ABB RAPID module: Module1.mod

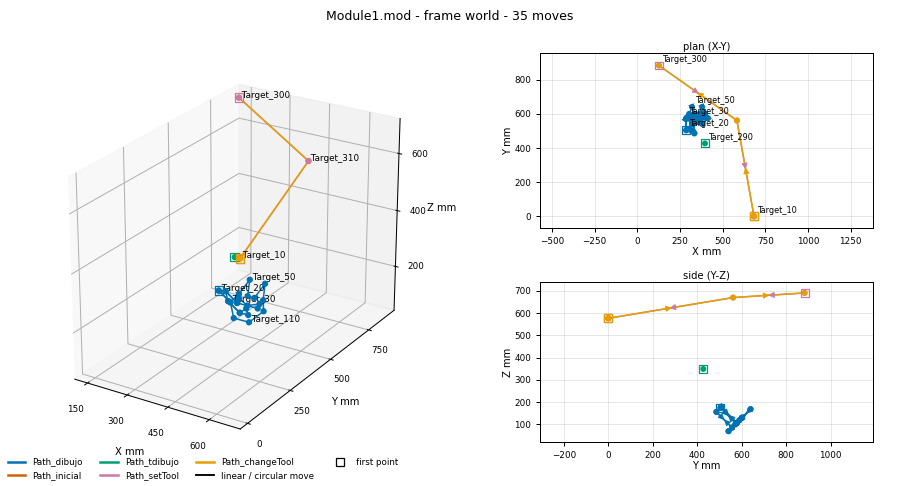
[picture p0: tool path of Module1.mod in frame world, 35 of 35 moves have a stored position in this frame; points joined in program order, loops and branches not executed]
MODULE Module1
        CONST robtarget Target_20:=[[-143.869244178,87.031135529,-100.000191842],[0.335710695,0,0,-0.941965142],[0,0,0,0],[9E+09,9E+09,9E+09,9E+09,9E+09,9E+09]];
    CONST robtarget Target_30:=[[-143.869244206,87.031135529,-0.000191841],[0.335710695,0,0,-0.941965142],[0,0,0,0],[9E+09,9E+09,9E+09,9E+09,9E+09,9E+09]];
    CONST robtarget Target_40:=[[-108.026112862,104.235837146,-0.000191832],[0.335710695,0,0,-0.941965142],[0,0,0,0],[9E+09,9E+09,9E+09,9E+09,9E+09,9E+09]];
    CONST robtarget Target_50:=[[-52.110827945,121.440538768,-0.000191815],[0.335710694,0,0.000000001,-0.941965143],[0,0,0,0],[9E+09,9E+09,9E+09,9E+09,9E+09,9E+09]];
    CONST robtarget Target_60:=[[-108.026112855,137.808909158,-0.000191832],[0.335710694,0,0.000000001,-0.941965143],[0,0,0,0],[9E+09,9E+09,9E+09,9E+09,9E+09,9E+09]];
    CONST robtarget Target_70:=[[-108.026112855,163.915610617,-0.000191832],[0.335710695,0,0,-0.941965142],[0,0,0,0],[9E+09,9E+09,9E+09,9E+09,9E+09,9E+09]];
    CONST robtarget Target_80:=[[-52.110827945,180.283981007,-0.000191815],[0.335710695,0,-0.000000001,-0.941965142],[0,0,0,0],[9E+09,9E+09,9E+09,9E+09,9E+09,9E+09]];
    CONST robtarget Target_90:=[[-108.026112862,197.48868263,-0.000191832],[0.335710695,0,-0.000000001,-0.941965142],[0,0,0,0],[9E+09,9E+09,9E+09,9E+09,9E+09,9E+09]];
    CONST robtarget Target_100:=[[-143.869244206,214.693384246,-0.000191841],[0.335710695,0,0,-0.941965142],[0,0,0,0],[9E+09,9E+09,9E+09,9E+09,9E+09,9E+09]];
    CONST robtarget Target_110:=[[-192.615902843,180.283981007,-0.000191856],[0.335710695,0,0,-0.941965142],[0,0,0,0],[9E+09,9E+09,9E+09,9E+09,9E+09,9E+09]];
    CONST robtarget Target_120:=[[-192.615902844,121.440538769,-0.000191855],[0.335710695,0,0,-0.941965142],[0,0,0,0],[9E+09,9E+09,9E+09,9E+09,9E+09,9E+09]];
    CONST robtarget Target_130:=[[-143.869244206,87.031135529,-0.000191841],[0.335710695,0,0,-0.941965142],[0,0,0,0],[9E+09,9E+09,9E+09,9E+09,9E+09,9E+09]];
    CONST robtarget Target_140:=[[-143.869244178,87.031135529,-100.000191842],[0.335710695,0,0,-0.941965142],[0,0,0,0],[9E+09,9E+09,9E+09,9E+09,9E+09,9E+09]];
    CONST robtarget Target_150:=[[-139.856817565,111.33818796,-100.000191841],[0.335710706,0,0,-0.941965138],[0,0,0,0],[9E+09,9E+09,9E+09,9E+09,9E+09,9E+09]];
    CONST robtarget Target_160:=[[-139.856817593,111.33818796,-0.00019184],[0.335710706,0,0,-0.941965138],[0,0,0,0],[9E+09,9E+09,9E+09,9E+09,9E+09,9E+09]];
    CONST robtarget Target_170:=[[-123.434971754,111.33818796,-0.000191836],[0.335710706,0,0,-0.941965138],[0,0,0,0],[9E+09,9E+09,9E+09,9E+09,9E+09,9E+09]];
    CONST robtarget Target_180:=[[-139.282664103,150.862259888,-0.000191841],[0.335710706,-0.000000001,-0.000000001,-0.941965138],[0,0,0,0],[9E+09,9E+09,9E+09,9E+09,9E+09,9E+09]];
    CONST robtarget Target_190:=[[-123.434971754,190.386331815,-0.000191836],[0.335710706,0,0.000000001,-0.941965138],[0,0,0,0],[9E+09,9E+09,9E+09,9E+09,9E+09,9E+09]];
    CONST robtarget Target_200:=[[-139.856817593,190.386331815,-0.00019184],[0.335710706,0,0,-0.941965138],[0,0,0,0],[9E+09,9E+09,9E+09,9E+09,9E+09,9E+09]];
    CONST robtarget Target_210:=[[-139.856817593,111.33818796,-0.00019184],[0.335710706,0,0,-0.941965138],[0,0,0,0],[9E+09,9E+09,9E+09,9E+09,9E+09,9E+09]];
    CONST robtarget Target_220:=[[-139.856817565,111.33818796,-100.000191841],[0.335710706,0,0,-0.941965138],[0,0,0,0],[9E+09,9E+09,9E+09,9E+09,9E+09,9E+09]];
    CONST robtarget Target_230:=[[-169.742573497,134.622057219,-100.000191849],[0.335710706,0,0,-0.941965138],[0,0,0,0],[9E+09,9E+09,9E+09,9E+09,9E+09,9E+09]];
    CONST robtarget Target_240:=[[-169.742573525,134.622057219,-0.000191849],[0.335710706,0,0,-0.941965138],[0,0,0,0],[9E+09,9E+09,9E+09,9E+09,9E+09,9E+09]];
    CONST robtarget Target_250:=[[-150.103708423,150.862259887,-0.000191843],[0.335710706,0,0,-0.941965138],[0,0,0,0],[9E+09,9E+09,9E+09,9E+09,9E+09,9E+09]];
    CONST robtarget Target_260:=[[-169.742573525,167.102462557,-0.000191849],[0.335710706,0,0,-0.941965138],[0,0,0,0],[9E+09,9E+09,9E+09,9E+09,9E+09,9E+09]];
    CONST robtarget Target_270:=[[-169.742573525,134.622057219,-0.000191849],[0.335710706,0,0,-0.941965138],[0,0,0,0],[9E+09,9E+09,9E+09,9E+09,9E+09,9E+09]];
    CONST robtarget Target_280:=[[-169.742573497,134.622057219,-100.000191849],[0.335710706,0,0,-0.941965138],[0,0,0,0],[9E+09,9E+09,9E+09,9E+09,9E+09,9E+09]];
    CONST robtarget Target_10:=[[683.826857055,0,576.999996593],[0.499999994,0,0.866025407,0],[0,0,0,0],[9E+09,9E+09,9E+09,9E+09,9E+09,9E+09]];
    CONST robtarget Target_290:=[[396.786283568,427.182015311,348.94513545],[0.291756838,-0.37886731,0.868997985,0.127200673],[0,0,-1,0],[9E+09,9E+09,9E+09,9E+09,9E+09,9E+09]];
    CONST robtarget Target_300:=[[127.426507212,883.161303543,691.12368836],[0.534755638,-0.462711495,0.534265162,0.463136282],[0,0,-1,0],[9E+09,9E+09,9E+09,9E+09,9E+09,9E+09]];
    CONST robtarget Target_310:=[[583.778205669,561.321662028,670.301501814],[0.628669244,-0.274711631,0.682050295,0.25321117],[0,-1,0,0],[9E+09,9E+09,9E+09,9E+09,9E+09,9E+09]];
!------------------------
    PROC main()
        Path_inicial;
    	WaitTime 1;
        IF DI_01 = 1 THEN
            SetDO DO_01,1;
            Path_tdibujo;
            Path_dibujo;
            Path_tdibujo;
            Path_inicial;
        ELSEIF DI_02 = 1 THEN
            Path_changeTool;
            SetDO DO_01,0;
            WaitDI DI_02,1;
            Path_setTool;
        ELSE
            Path_inicial;
        ENDIF
    ENDPROC
    PROC Path_dibujo()
        MoveL Target_20,v200,z5,ToolMarker\WObj:=W_Board;
        MoveL Target_30,v200,z5,ToolMarker\WObj:=W_Board;
        MoveL Target_40,v200,z5,ToolMarker\WObj:=W_Board;
        MoveL Target_50,v200,z5,ToolMarker\WObj:=W_Board;
        MoveL Target_60,v200,z5,ToolMarker\WObj:=W_Board;
        MoveL Target_70,v200,z5,ToolMarker\WObj:=W_Board;
        MoveL Target_80,v200,z5,ToolMarker\WObj:=W_Board;
        MoveL Target_90,v200,z5,ToolMarker\WObj:=W_Board;
        MoveL Target_100,v200,z5,ToolMarker\WObj:=W_Board;
        MoveL Target_110,v200,z5,ToolMarker\WObj:=W_Board;
        MoveL Target_120,v200,z5,ToolMarker\WObj:=W_Board;
        MoveL Target_130,v200,z5,ToolMarker\WObj:=W_Board;
        MoveL Target_140,v200,z5,ToolMarker\WObj:=W_Board;
        MoveL Target_150,v200,z5,ToolMarker\WObj:=W_Board;
        MoveL Target_160,v200,z5,ToolMarker\WObj:=W_Board;
        MoveL Target_170,v200,z5,ToolMarker\WObj:=W_Board;
        MoveL Target_180,v200,z5,ToolMarker\WObj:=W_Board;
        MoveL Target_190,v200,z5,ToolMarker\WObj:=W_Board;
        MoveL Target_200,v200,z5,ToolMarker\WObj:=W_Board;
        MoveL Target_210,v200,z5,ToolMarker\WObj:=W_Board;
        MoveL Target_220,v200,z5,ToolMarker\WObj:=W_Board;
        MoveL Target_230,v200,z5,ToolMarker\WObj:=W_Board;
        MoveL Target_240,v200,z5,ToolMarker\WObj:=W_Board;
        MoveL Target_250,v200,z5,ToolMarker\WObj:=W_Board;
        MoveL Target_260,v200,z5,ToolMarker\WObj:=W_Board;
        MoveL Target_270,v200,z5,ToolMarker\WObj:=W_Board;
        MoveL Target_280,v200,z5,ToolMarker\WObj:=W_Board;
    ENDPROC
    PROC Path_inicial()
        MoveJ Target_10,v400,z100,ToolMarker\WObj:=wobj0;
    ENDPROC
    PROC Path_tdibujo()
        MoveL Target_290,v400,z100,ToolMarker\WObj:=wobj0;
    ENDPROC
    PROC Path_setTool()
        MoveL Target_300,v1000,z100,ToolMarker\WObj:=wobj0;
        MoveL Target_310,v1000,z100,ToolMarker\WObj:=wobj0;
        MoveL Target_10,v1000,z100,ToolMarker\WObj:=wobj0;
    ENDPROC
    PROC Path_changeTool()
        MoveL Target_10,v1000,z100,ToolMarker\WObj:=wobj0;
        MoveL Target_310,v1000,z100,ToolMarker\WObj:=wobj0;
        MoveL Target_300,v1000,z100,ToolMarker\WObj:=wobj0;
    ENDPROC
ENDMODULE
